Staubli VAL3: init.pgx

public program init()
  local num l_nStatus
begin
  // Copyright (c) 2021, Institute for Factory Automation and Production Systems (FAPS)
  //
  // Licensed under the Apache License, Version 2.0 (the "License");
  // you may not use this file except in compliance with the License.
  // You may obtain a copy of the License at
  //
  //     http://www.apache.org/licenses/LICENSE-2.0
  //
  // Unless required by applicable law or agreed to in writing, software
  // distributed under the License is distributed on an "AS IS" BASIS,
  // WITHOUT WARRANTIES OR CONDITIONS OF ANY KIND, either express or implied.
  // See the License for the specific language governing permissions and
  // limitations under the License.


  logMsg("[INFO] Called IOInterface:init()")

  // init IOModule enum
  call IOModule:init()

  // check IO status of the BasicIO module
  l_nStatus = ioStatus(diBasicIn[0])
  if (l_nStatus >= 0)
    bBasicIO1=true
    logMsg("[INFO] BasicIO available (status: "+toString("", l_nStatus)+")")
  else
    bBasicIO1=false
    logMsg("[INFO] BasicIO not available (status: "+toString("", l_nStatus)+")")
  endIf

  // check IO status of the BasicIO-2 module
  l_nStatus = ioStatus(diBasicIn2[0])
  if (l_nStatus >= 0)
    bBasicIO2=true
    logMsg("[INFO] BasicIO-2 available (status: "+toString("", l_nStatus)+")")
  else
    bBasicIO2=false
    logMsg("[INFO] BasicIO-2 not available (status: "+toString("", l_nStatus)+")")
  endIf
end
